// TwinCAT 3 PLC project PLC
// Title: Test PLC project for ads-client library
// Company: Jussi Isotalo
// Author: Jussi Isotalo
// Description: Copyright (c) 2022 Jussi Isotalo <j.isotalo91@gmail.com> Permission is hereby granted, free of charge, to any person obtaining a copy of this software and associated documentation files (the "Software"), to deal in the Software without restriction, including without limitation the rights to use, copy, modify, merge, publish, distribute, sublicense, and/or sell copies of the Software, and to permit persons to whom the Software is furnished to do so, subject to the following conditions: The above copyright notice and this permission notice shall be included in all copies or substantial portions of the Software. THE SOFTWARE IS PROVIDED "AS IS", WITHOUT WARRANTY OF ANY KIND, EXPRESS OR IMPLIED, INCLUDING BUT NOT LIMITED TO THE WARRANTIES OF MERCHANTABILITY, FITNESS FOR A PARTICULAR PURPOSE AND NONINFRINGEMENT. IN NO EVENT SHALL THE AUTHORS OR COPYRIGHT HOLDERS BE LIABLE FOR ANY CLAIM, DAMAGES OR OTHER LIABILITY, WHETHER IN AN ACTION OF CONTRACT, TORT OR OTHERWISE, ARISING FROM, OUT OF OR IN CONNECTION WITH THE SOFTWARE OR THE USE OR OTHER DEALINGS IN THE SOFTWARE
// ProgramVersion: 3.1.4023.0
// libraries:
//   Tc2_DataExchange, * (Beckhoff Automation GmbH)
//   Tc2_Standard, * (Beckhoff Automation GmbH)
//   Tc2_System, * (Beckhoff Automation GmbH)
//   Tc2_Utilities, * (Beckhoff Automation GmbH)
//   Tc3_Module, * (Beckhoff Automation GmbH)
// project tree:
//   AdsClientTests/Data types/ E_ExtendedEnum.TcDUT, FB_Block.TcPOU, FB_EmptyBlock.TcPOU, FB_EmptyBlock_1.TcPOU, I_Interface.TcIO, ST_Bits.TcDUT, ST_ComplexTypes_PackMode1.TcDUT, ST_ComplexTypes_PackMode8.TcDUT, ST_EmptyStruct.TcDUT, ST_IssueSpecificTypes.TcDUT, ST_SpecialTypes.TcDUT, ST_StandardTypes_PackMode1.TcDUT, ST_StandardTypes_PackMode8.TcDUT, ST_ComplexArrayTypes.TcDUT, ST_Struct.TcDUT, E_Enum.TcDUT, E_LintEnum.TcDUT, StandardTypesAlias.TcDUT, ST_StandardTypes.TcDUT, ST_StandardArrayTypes.TcDUT, ST_ComplexTypes.TcDUT, U_Union.TcDUT
//   AdsClientTests/ GVL_AdsClientTests.TcGVL, PRG_AdsClientTests.TcPOU
//   AdsClientTests/Read/ GVL_Read.TcGVL
//   AdsClientTests/RPC/ FB_Rpc.TcPOU, GVL_RPC.TcGVL
//   AdsClientTests/Subscription/ GVL_Subscription.TcGVL, PRG_Subscription.TcPOU
//   AdsClientTests/Symbols and datatypes/ GVL_SymbolsAndDataTypes.TcGVL, ST_TestDataType.TcDUT
//   AdsClientTests/Write/ GVL_Write.TcGVL
//   AdsClientTests/_OLD/ ST_Issue94.TcDUT, ST_Issue94_Byte.TcDUT, ST_PackMode1.TcDUT, ST_PackMode8.TcDUT, ST_Struct2.TcDUT
//   / PlcTask.TcTTO
// real-time tasks:
//   TASK PlcTask: cycle T#10ms, priority 20, ADS port 350
//   TASK PlcTask_852: cycle T#10ms, priority 21, ADS port 351

CONFIGURATION PLC
    RESOURCE PLC ON TwinCAT3
        TASK PlcTask(INTERVAL := T#10ms, PRIORITY := 20);
        PROGRAM PRG_AdsClientTests WITH PlcTask : PRG_AdsClientTests;
    END_RESOURCE
END_CONFIGURATION

// ---- AdsClientTests/Data types/E_ExtendedEnum.TcDUT
{attribute 'qualified_only'}
//{attribute 'strict'}
//This enum works differently than E_Enum only on TC 4026 and newer (comments and attributes)
TYPE E_ExtendedEnum :
(
	Disabled 	:= 0, //Machine is disabled
	Starting 	:= 50, //Machine is starting
	Running 	:= 100, //Machine is running
	Stopping	:= 200, //Machine is stopping
	
	{attribute 'ads-client-enum-attribute' := 'example-enum-value-ääö'}
	Unknown		:= -99 //Machine is ääöööÄÄÖö
);
END_TYPE

// ---- AdsClientTests/Data types/ST_Bits.TcDUT
TYPE ST_Bits :
STRUCT
	Bit_0 : BIT := TRUE;
	Bit_1 : BIT := FALSE;
	Bit_2 : BIT := FALSE;
	Bit_3 : BIT := TRUE;
	Bit_4 : BIT := TRUE;
	Bit_5 : BIT := FALSE;
	Bit_6 : BIT := FALSE;
	Bit_7 : BIT := TRUE;
	
	Bit_8 : BIT := FALSE;
	Bit_9 : BIT := TRUE;
	Bit_10 : BIT := TRUE;
	Bit_11 : BIT := FALSE;
	Bit_12 : BIT := FALSE;
	Bit_13 : BIT := TRUE;
	Bit_14 : BIT := TRUE;
	Bit_15 : BIT := FALSE;
	
	REAL_ : REAL := 3.14;
	
	Bit_16 : BIT := TRUE;
	Bit_17 : BIT := TRUE;
	Bit_18 : BIT := FALSE;
	Bit_19 : BIT := TRUE;
	Bit_20 : BIT := TRUE;
	Bit_21 : BIT := FALSE;
	Bit_22 : BIT := FALSE;
	Bit_23 : BIT := TRUE;
	
	Bit_24 : BIT := TRUE;
	Bit_25 : BIT := FALSE;
	Bit_26 : BIT := TRUE;
	Bit_27 : BIT := TRUE;
	Bit_28 : BIT := FALSE;
	Bit_29 : BIT := TRUE;
	Bit_30 : BIT := TRUE;
	Bit_31 : BIT := FALSE;
	
	Bit_32 : BIT := TRUE;
END_STRUCT
END_TYPE

// ---- AdsClientTests/Data types/ST_ComplexTypes_PackMode1.TcDUT
{attribute 'pack_mode' := '1'}
TYPE ST_ComplexTypes_PackMode1 :
STRUCT
	STRUCT_ 	: ST_StandardTypes;
	STRUCT_2 	: ST_StandardArrayTypes;
	ALIAS_ 		: StandardTypesAlias;
	ENUM_		: E_Enum := E_Enum.Running;
	ENUM_2		: E_Enum := E_Enum.Unknown;
	ENUM_3		: E_Enum := 5555; //Not a valid value
	ENUM_4		: E_LintEnum := E_LintEnum.Negative;
	ENUM_5		: (Implicit, Enum, Values, Go, Here) := Values;
	POINTER_	: POINTER TO ST_StandardTypes;
	REFERENCE_	: REFERENCE TO ST_StandardTypes;
	SUBRANGE_	: INT(-4095..4095) := 1234;
	UNION_		: U_Union := (STRING_ := 'A test string ääöö!!@@'); 
	UNION_2		: U_Union := (INT_ := 32767); 
	UNION_3		: U_Union := (REAL_ := 3.14);
	BLOCK_		: FB_Block;
	BLOCK_2		: TON := (PT := T#2S500MS);
	BLOCK_3		: TC2_System.FB_CreateDir := (sPathName := 'C:\Test');
	BLOCK_4		: Tc2_DataExchange.FB_ReadAdsSymByName := (sVarName := 'GVL_Test.Variable');
	INTERFACE_	: I_Interface := BLOCK_;
END_STRUCT
END_TYPE

// ---- AdsClientTests/Data types/ST_ComplexTypes_PackMode8.TcDUT
{attribute 'pack_mode' := '1'}
TYPE ST_ComplexTypes_PackMode8 :
STRUCT
	STRUCT_ 	: ST_StandardTypes;
	STRUCT_2 	: ST_StandardArrayTypes;
	ALIAS_ 		: StandardTypesAlias;
	ENUM_		: E_Enum := E_Enum.Running;
	ENUM_2		: E_Enum := E_Enum.Unknown;
	ENUM_3		: E_Enum := 5555; //Not a valid value
	ENUM_4		: E_LintEnum := E_LintEnum.Negative;
	ENUM_5		: (Implicit, Enum, Values, Go, Here) := Values;
	POINTER_	: POINTER TO ST_StandardTypes;
	REFERENCE_	: REFERENCE TO ST_StandardTypes;
	SUBRANGE_	: INT(-4095..4095) := 1234;
	UNION_		: U_Union := (STRING_ := 'A test string ääöö!!@@'); 
	UNION_2		: U_Union := (INT_ := 32767); 
	UNION_3		: U_Union := (REAL_ := 3.14);
	BLOCK_		: FB_Block;
	BLOCK_2		: TON := (PT := T#2S500MS);
	BLOCK_3		: TC2_System.FB_CreateDir := (sPathName := 'C:\Test');
	BLOCK_4		: Tc2_DataExchange.FB_ReadAdsSymByName := (sVarName := 'GVL_Test.Variable');
	INTERFACE_	: I_Interface := BLOCK_;
END_STRUCT
END_TYPE

// ---- AdsClientTests/Data types/ST_EmptyStruct.TcDUT
TYPE ST_EmptyStruct :
STRUCT
END_STRUCT
END_TYPE

// ---- AdsClientTests/Data types/ST_IssueSpecificTypes.TcDUT
TYPE ST_IssueSpecificTypes :
STRUCT
	Issue94	: ST_Issue94;
END_STRUCT
END_TYPE

// ---- AdsClientTests/Data types/ST_SpecialTypes.TcDUT
TYPE ST_SpecialTypes :
STRUCT
	NegativeIndexArray		: ARRAY[-100..100] OF LREAL := [1.11, 99(0.0), 5.55, 99(0.0), 9.99];
	MultiDimensionalArray	: ARRAY[1..3, 1..2] OF BYTE := [1, 2, 3, 4, 5, 6];
	ArrayOfArrays			: ARRAY[1..3] OF ARRAY[1..2] OF SINT := [[-1, -2], [-3, -4], [-5, -6]];
	
	PackMode1		: ST_StandardTypes_PackMode1;
	PackMode1_2		: ST_ComplexTypes_PackMode1;
	PackMode8		: ST_StandardTypes_PackMode8;
	PackMode8_2		: ST_ComplexTypes_PackMode8;
	
	EmptyBlock		: FB_EmptyBlock;
	EmptyStruct		: ST_EmptyStruct;
	EmptyArray 		: ARRAY[0..-1] OF BOOL; //How is this even possible..?
	
	Bits			: ST_Bits;
	
    {attribute 'TcEncoding':='UTF-8'}
	STRING_UTF8		: STRING := 'A test string ääöö!!@@';
END_STRUCT
END_TYPE

// ---- AdsClientTests/Data types/ST_StandardTypes_PackMode1.TcDUT
{attribute 'pack_mode' := '1'}
TYPE ST_StandardTypes_PackMode1 :
STRUCT
	BOOL_ 	: BOOL := TRUE;
	BOOL_2 	: BOOL := FALSE;
	BYTE_ 	: BYTE := 255;
	WORD_ 	: WORD := 65535;
	DWORD_ 	: DWORD := 4294967295;
	SINT_ 	: SINT := 127;
	SINT_2 	: SINT := -128;
	USINT_ 	: USINT := 255;
	INT_ 	: INT := 32767;
	INT_2 	: INT := -32768;
	UINT_ 	: UINT := 65535;
	DINT_ 	: DINT := 2147483647;
	DINT_2 	: DINT := -2147483648;
	UDINT_ 	: UDINT := 4294967295;
	REAL_ 	: REAL := 3.4E38;
	REAL_2 	: REAL := -3.4E38;
	REAL_3 	: REAL := 75483.545;
	REAL_4 	: REAL := -75483.545;
	STRING_	: STRING := 'A test string ääöö!!@@';
	STRING_2: STRING(255) := 'Lorem ipsum dolor sit amet, consectetur adipiscing elit. Pellentesque bibendum mauris vel metus rutrum, sed gravida justo dignissim. Aenean et nisi cursus, auctor mi vel, posuere enim. Suspendisse ultricies mauris in finibus tristique. Nullam turpis duis.';
	DATE_ 	: DATE := D#2106-02-06;
	DT_ 	: DT := DT#2106-02-06-06:28:15;
	DT_2 	: DATE_AND_TIME := DT#2106-02-06-06:28:15;
	TOD_ 	: TOD := TO_TOD(4294967295);
	TOD_2 	: TIME_OF_DAY := TO_TOD(4294967295);
	TIME_ 	: TIME := T#49D17H2M47S295MS;
	LWORD_	: LWORD := 18446744073709551615;
	LINT_	: LINT := 9223372036854775807;
	LINT_2	: LINT := -9223372036854775808;
	ULINT_	: ULINT := 18446744073709551615;
	LREAL_ 	: LREAL := 1.7E308;
	LREAL_2 : LREAL := -1.7E308;
	LREAL_3 : REAL := 75483.545;
	LREAL_4 : REAL := -75483.545;
	WSTRING_: WSTRING := "A test wstring ääöö!!@@ ẞẟΔش";
	WSTRING_2: WSTRING(255) := "Lorem ipsum dolor sit amet, consectetur adipiscing elit. Pellentesque bibendum mauris vel metus rutrum, sed gravida justo dignissim. Aenean et nisi cursus, auctor mi vel, posuere enim. Suspendisse ultricies mauris in finibus tristique. Nullam turpis duis.";
	//LDATE_	: LDATE := LD#2554-7-21;
	//LDT_	: LDT := LDT#2554-7-21-23:34:33.709551615;
	//LTOD_	: LTOD := LTOD#23:59:59.999999999;
	LTIME_ 	: LTIME := LTIME#213503D23H34M33S709MS551US615NS;
END_STRUCT
END_TYPE

// ---- AdsClientTests/Data types/ST_StandardTypes_PackMode8.TcDUT
{attribute 'pack_mode' := '8'}
TYPE ST_StandardTypes_PackMode8:
STRUCT
	BOOL_ 	: BOOL := TRUE;
	BOOL_2 	: BOOL := FALSE;
	BYTE_ 	: BYTE := 255;
	WORD_ 	: WORD := 65535;
	DWORD_ 	: DWORD := 4294967295;
	SINT_ 	: SINT := 127;
	SINT_2 	: SINT := -128;
	USINT_ 	: USINT := 255;
	INT_ 	: INT := 32767;
	INT_2 	: INT := -32768;
	UINT_ 	: UINT := 65535;
	DINT_ 	: DINT := 2147483647;
	DINT_2 	: DINT := -2147483648;
	UDINT_ 	: UDINT := 4294967295;
	REAL_ 	: REAL := 3.4E38;
	REAL_2 	: REAL := -3.4E38;
	REAL_3 	: REAL := 75483.545;
	REAL_4 	: REAL := -75483.545;
	STRING_	: STRING := 'A test string ääöö!!@@';
	STRING_2: STRING(255) := 'Lorem ipsum dolor sit amet, consectetur adipiscing elit. Pellentesque bibendum mauris vel metus rutrum, sed gravida justo dignissim. Aenean et nisi cursus, auctor mi vel, posuere enim. Suspendisse ultricies mauris in finibus tristique. Nullam turpis duis.';
	DATE_ 	: DATE := D#2106-02-06;
	DT_ 	: DT := DT#2106-02-06-06:28:15;
	DT_2 	: DATE_AND_TIME := DT#2106-02-06-06:28:15;
	TOD_ 	: TOD := TO_TOD(4294967295);
	TOD_2 	: TIME_OF_DAY := TO_TOD(4294967295);
	TIME_ 	: TIME := T#49D17H2M47S295MS;
	LWORD_	: LWORD := 18446744073709551615;
	LINT_	: LINT := 9223372036854775807;
	LINT_2	: LINT := -9223372036854775808;
	ULINT_	: ULINT := 18446744073709551615;
	LREAL_ 	: LREAL := 1.7E308;
	LREAL_2 : LREAL := -1.7E308;
	LREAL_3 : REAL := 75483.545;
	LREAL_4 : REAL := -75483.545;
	WSTRING_: WSTRING := "A test wstring ääöö!!@@ ẞẟΔش";
	WSTRING_2: WSTRING(255) := "Lorem ipsum dolor sit amet, consectetur adipiscing elit. Pellentesque bibendum mauris vel metus rutrum, sed gravida justo dignissim. Aenean et nisi cursus, auctor mi vel, posuere enim. Suspendisse ultricies mauris in finibus tristique. Nullam turpis duis.";
	//LDATE_	: LDATE := LD#2554-7-21;
	//LDT_	: LDT := LDT#2554-7-21-23:34:33.709551615;
	//LTOD_	: LTOD := LTOD#23:59:59.999999999;
	LTIME_ 	: LTIME := LTIME#213503D23H34M33S709MS551US615NS;
END_STRUCT
END_TYPE

// ---- AdsClientTests/Data types/ST_ComplexArrayTypes.TcDUT
TYPE ST_ComplexArrayTypes :
STRUCT
	STRUCT_ 	: ARRAY[0..2] OF ST_StandardTypes;
	STRUCT_2 	: ARRAY[0..2] OF ST_StandardArrayTypes;
	ALIAS_ 		: ARRAY[0..2] OF StandardTypesAlias;
	ENUM_		: ARRAY[0..2] OF E_Enum := [E_Enum.Running, E_Enum.Disabled, E_Enum.Stopping];
	ENUM_2		: ARRAY[0..2] OF E_Enum := [E_Enum.Unknown, E_Enum.Disabled, E_Enum.Starting];
	ENUM_3		: ARRAY[0..2] OF E_Enum := [5555, 0, E_Enum.Unknown];
	ENUM_4		: ARRAY[0..2] OF E_LintEnum := [E_LintEnum.Negative, E_LintEnum.Zero, E_LintEnum.Positive];
	ENUM_5		: ARRAY[0..2] OF (Implicit, Enum, Values, Go, Here) := [2, 0, 4];
	POINTER_	: ARRAY[0..2] OF POINTER TO ST_StandardTypes;
	//REFERENCE_	: ARRAY[0..2] OF REFERENCE TO ST_StandardTypes;
	SUBRANGE_	: ARRAY[0..2] OF INT(-4095..4095) := [1234, 0, -1234];
	UNION_		: ARRAY[0..2] OF U_Union := [
		(STRING_ := 'A test string ääöö!!@@'),
		(INT_ := 32767),
		(REAL_ := 3.14)
	]; 
	BLOCK_		: ARRAY[0..2] OF FB_Block := [
		(StrValue := 'First'),
		(),
		(StrValue := 'Third')
	];
	BLOCK_2		: ARRAY[0..2] OF TON := [(PT := T#2S500MS), (), (PT := T#123S)];
	BLOCK_3		: ARRAY[0..2] OF TC2_System.FB_CreateDir := [
		(sPathName := 'C:\Test'),
		(),
		(sPathName := 'C:\AnotherTest')
	];
	BLOCK_4		: ARRAY[0..2] OF Tc2_DataExchange.FB_ReadAdsSymByName := [
		(sVarName := 'GVL_Test.Variable'),
		(),
		(sVarName := 'GVL_Test.AnotherVariable')
	];
	INTERFACE_	: ARRAY[0..2] OF I_Interface := [BLOCK_[0], 0, BLOCK_[2]];
END_STRUCT
END_TYPE

// ---- AdsClientTests/Data types/ST_Struct.TcDUT
TYPE ST_Struct :
STRUCT
	SomeText : STRING(50) := 'Hello ads-client';
	SomeReal : REAL := 3.14159265359;
	SomeDate : DT := DT#2020-4-13-12:25:33;
END_STRUCT
END_TYPE

// ---- AdsClientTests/Symbols and datatypes/ST_TestDataType.TcDUT
{attribute 'pack_mode' := '3'}
{attribute 'ads-client-datatype-attribute' := 'example-datatype-value-ääö'}
//Test comment äääöö 
TYPE ST_TestDataType :
STRUCT
	Member : ST_Struct;
END_STRUCT
END_TYPE

// ---- AdsClientTests/Data types/E_Enum.TcDUT
{attribute 'qualified_only'}
//{attribute 'strict'}
TYPE E_Enum :
(
	Disabled 	:= 0,
	Starting 	:= 50,
	Running 	:= 100,
	Stopping	:= 200,
	Unknown		:= -99
);
END_TYPE

// ---- AdsClientTests/Data types/E_LintEnum.TcDUT
{attribute 'qualified_only'}
//{attribute 'strict'}
TYPE E_LintEnum :
(
	Negative := -9223372036854775808,
	Zero := 0,
	Positive := 9223372036854775807
) LINT;
END_TYPE

// ---- AdsClientTests/Data types/StandardTypesAlias.TcDUT
TYPE StandardTypesAlias : ST_StandardTypes; END_TYPE

// ---- AdsClientTests/Data types/ST_StandardTypes.TcDUT
TYPE ST_StandardTypes :
STRUCT
	BOOL_ 	: BOOL := TRUE;
	BOOL_2 	: BOOL := FALSE;
	BYTE_ 	: BYTE := 255;
	WORD_ 	: WORD := 65535;
	DWORD_ 	: DWORD := 4294967295;
	SINT_ 	: SINT := 127;
	SINT_2 	: SINT := -128;
	USINT_ 	: USINT := 255;
	INT_ 	: INT := 32767;
	INT_2 	: INT := -32768;
	UINT_ 	: UINT := 65535;
	DINT_ 	: DINT := 2147483647;
	DINT_2 	: DINT := -2147483648;
	UDINT_ 	: UDINT := 4294967295;
	REAL_ 	: REAL := 3.4E38;
	REAL_2 	: REAL := -3.4E38;
	REAL_3 	: REAL := 75483.545;
	REAL_4 	: REAL := -75483.545;
	STRING_	: STRING := 'A test string ääöö!!@@';
	STRING_2: STRING(255) := 'Lorem ipsum dolor sit amet, consectetur adipiscing elit. Pellentesque bibendum mauris vel metus rutrum, sed gravida justo dignissim. Aenean et nisi cursus, auctor mi vel, posuere enim. Suspendisse ultricies mauris in finibus tristique. Nullam turpis duis.';
	DATE_ 	: DATE := D#2106-02-06;
	DT_ 	: DT := DT#2106-02-06-06:28:15;
	DT_2 	: DATE_AND_TIME := DT#2106-02-06-06:28:15;
	TOD_ 	: TOD := TO_TOD(4294967295);
	TOD_2 	: TIME_OF_DAY := TO_TOD(4294967295);
	TIME_ 	: TIME := T#49D17H2M47S295MS;
	LWORD_	: LWORD := 18446744073709551615;
	LINT_	: LINT := 9223372036854775807;
	LINT_2	: LINT := -9223372036854775808;
	ULINT_	: ULINT := 18446744073709551615;
	LREAL_ 	: LREAL := 1.7E308;
	LREAL_2 : LREAL := -1.7E308;
	LREAL_3 : REAL := 75483.545;
	LREAL_4 : REAL := -75483.545;
	WSTRING_: WSTRING := "A test wstring ääöö!!@@ ẞẟΔش";
	WSTRING_2: WSTRING(255) := "Lorem ipsum dolor sit amet, consectetur adipiscing elit. Pellentesque bibendum mauris vel metus rutrum, sed gravida justo dignissim. Aenean et nisi cursus, auctor mi vel, posuere enim. Suspendisse ultricies mauris in finibus tristique. Nullam turpis duis.";
	//LDATE_	: LDATE := LD#2554-7-21;
	//LDT_	: LDT := LDT#2554-7-21-23:34:33.709551615;
	//LTOD_	: LTOD := LTOD#23:59:59.999999999;
	LTIME_ 	: LTIME := LTIME#213503D23H34M33S709MS551US615NS;
END_STRUCT
END_TYPE

// ---- AdsClientTests/Data types/ST_StandardArrayTypes.TcDUT
TYPE ST_StandardArrayTypes :
STRUCT
	BOOL_ 	: ARRAY[0..2] OF BOOL := [TRUE, FALSE, TRUE];
	BOOL_2 	: ARRAY[0..2] OF BOOL := [FALSE, TRUE, FALSE];
	BYTE_ 	: ARRAY[0..2] OF BYTE := [255, 254, 0];
	WORD_ 	: ARRAY[0..2] OF WORD := [65535, 65534, 0];
	DWORD_ 	: ARRAY[0..2] OF DWORD := [4294967295, 4294967294, 0];
	SINT_ 	: ARRAY[0..2] OF SINT := [127, 126, 0];
	SINT_2 	: ARRAY[0..2] OF SINT := [-128, -127, 0];
	USINT_ 	: ARRAY[0..2] OF USINT := [255, 254, 0];
	INT_ 	: ARRAY[0..2] OF INT := [32767, 0, -32768];
	INT_2 	: ARRAY[0..2] OF INT := [-32768, 0, 32767];
	UINT_ 	: ARRAY[0..2] OF UINT := [65535, 65534, 0];
	DINT_ 	: ARRAY[0..2] OF DINT := [2147483647, 0, -2147483648];
	DINT_2 	: ARRAY[0..2] OF DINT := [-2147483648, 0, 2147483647];
	UDINT_ 	: ARRAY[0..2] OF UDINT := [4294967295, 4294967294, 0];
	REAL_ 	: ARRAY[0..2] OF REAL := [3.4E38, 0, -3.4E38];
	REAL_2 	: ARRAY[0..2] OF REAL := [-3.4E38, 0, 3.4E38];
	REAL_3 	: ARRAY[0..2] OF REAL := [75483.545, 0, -75483.545];
	REAL_4 	: ARRAY[0..2] OF REAL := [-75483.545, 0, 75483.545];
	STRING_	: ARRAY[0..2] OF STRING := ['A test string ääöö!!@@', '', 'String value'];
	STRING_2: ARRAY[0..2] OF STRING(255) := [
		'Lorem ipsum dolor sit amet, consectetur adipiscing elit. Pellentesque bibendum mauris vel metus rutrum, sed gravida justo dignissim. Aenean et nisi cursus, auctor mi vel, posuere enim. Suspendisse ultricies mauris in finibus tristique. Nullam turpis duis.',
		'',
		'Proin tempor diam a felis fermentum, id molestie tortor pharetra. Phasellus condimentum rhoncus ultrices. Suspendisse ultricies nec neque quis sodales. In molestie vestibulum nulla eu gravida. Morbi orci ipsum, gravida elementum eros non, egestas egestas.'];
	DATE_ 	: ARRAY[0..2] OF DATE := [D#2106-02-06, D#2106-02-05, TO_DATE(0)];
	DT_ 	: ARRAY[0..2] OF DT := [DT#2106-02-06-06:28:15, DT#2106-02-06-06:28:14, TO_DT(0)];
	DT_2 	: ARRAY[0..2] OF DATE_AND_TIME := [DT#2106-02-06-06:28:15, DT#2106-02-06-06:28:14, TO_DT(0)];
	TOD_ 	: ARRAY[0..2] OF TOD := [TO_TOD(4294967295), TO_TOD(4294967294), TO_TOD(0)];
	TOD_2 	: ARRAY[0..2] OF TIME_OF_DAY := [TO_TOD(4294967295), TO_TOD(4294967294), TO_TOD(0)];
	TIME_ 	: ARRAY[0..2] OF TIME := [T#49D17H2M47S295MS, T#49D17H2M47S294MS, T#0S];
	LWORD_	: ARRAY[0..2] OF LWORD := [18446744073709551615, 18446744073709551614, 0];
	LINT_	: ARRAY[0..2] OF LINT := [9223372036854775807, 0, -9223372036854775808];
	LINT_2	: ARRAY[0..2] OF LINT := [-9223372036854775808, 0, 9223372036854775807];
	ULINT_	: ARRAY[0..2] OF ULINT := [18446744073709551615, 18446744073709551614, 0];
	LREAL_ 	: ARRAY[0..2] OF LREAL := [1.7E308, 0, -1.7E308];
	LREAL_2 : ARRAY[0..2] OF LREAL := [-1.7E308, 0, 1.7E308];
	LREAL_3	: ARRAY[0..2] OF REAL := [75483.545, 0, -75483.545];
	LREAL_4	: ARRAY[0..2] OF REAL := [-75483.545, 0, 75483.545];
	WSTRING_: ARRAY[0..2] OF WSTRING := ["A test wstring ääöö!!@@ ẞẟΔش", "", "ẞẟΔ"];
	WSTRING_2: ARRAY[0..2] OF WSTRING(255) := [
		"Lorem ipsum dolor sit amet, consectetur adipiscing elit. Pellentesque bibendum mauris vel metus rutrum, sed gravida justo dignissim. Aenean et nisi cursus, auctor mi vel, posuere enim. Suspendisse ultricies mauris in finibus tristique. Nullam turpis duis.",
		"",
		"Proin tempor diam a felis fermentum, id molestie tortor pharetra. Phasellus condimentum rhoncus ultrices. Suspendisse ultricies nec neque quis sodales. In molestie vestibulum nulla eu gravida. Morbi orci ipsum, gravida elementum eros non, egestas egestas."
	];
	//LDATE_	: ARRAY[0..2] OF LDATE := [LD#2554-7-21];
	//LDT_	: ARRAY[0..2] OF LDT := [LDT#2554-7-21-23:34:33.709551615];
	//LTOD_	: ARRAY[0..2] OF LTOD := [LTOD#23:59:59.999999999];
	LTIME_ 	: ARRAY[0..2] OF LTIME := [LTIME#213503D23H34M33S709MS551US615NS, LTIME#213503D23H34M33S709MS551US614NS, LTIME#0S];
END_STRUCT
END_TYPE

// ---- AdsClientTests/Data types/ST_ComplexTypes.TcDUT
TYPE ST_ComplexTypes :
STRUCT
	STRUCT_ 	: ST_StandardTypes;
	STRUCT_2 	: ST_StandardArrayTypes;
	ALIAS_ 		: StandardTypesAlias;
	ENUM_		: E_Enum := E_Enum.Running;
	ENUM_2		: E_Enum := E_Enum.Unknown;
	ENUM_3		: E_Enum := 5555; //Not a valid value
	ENUM_4		: E_LintEnum := E_LintEnum.Negative;
	ENUM_5		: (Implicit, Enum, Values, Go, Here) := Values;
	ENUM_6		: E_ExtendedEnum := E_Enum.Unknown;
	POINTER_	: POINTER TO ST_StandardTypes;
	REFERENCE_	: REFERENCE TO ST_StandardTypes;
	SUBRANGE_	: INT(-4095..4095) := 1234;
	UNION_		: U_Union := (STRING_ := 'A test string ääöö!!@@'); 
	UNION_2		: U_Union := (INT_ := 32767); 
	UNION_3		: U_Union := (REAL_ := 3.14);
	BLOCK_		: FB_Block;
	BLOCK_2		: TON := (PT := T#2S500MS);
	BLOCK_3		: TC2_System.FB_CreateDir := (sPathName := 'C:\Test');
	BLOCK_4		: Tc2_DataExchange.FB_ReadAdsSymByName := (sVarName := 'GVL_Test.Variable');
	INTERFACE_	: I_Interface := BLOCK_;
END_STRUCT
END_TYPE

// ---- AdsClientTests/Data types/U_Union.TcDUT
TYPE U_Union :
UNION
	INT_	: INT;
	BOOL_	: BOOL;
	UDINT_	: UDINT;
	STRING_	: STRING;
	REAL_	: REAL;
END_UNION
END_TYPE

// ---- AdsClientTests/_OLD/ST_Issue94.TcDUT
TYPE ST_Issue94 :
STRUCT
	BoolValue 	: bool := TRUE;
	ArrayValue 	:  ARRAY [0..1] OF ST_Issue94_Byte := [(ByteValue := 1), (ByteValue := 2)];
END_STRUCT
END_TYPE

// ---- AdsClientTests/_OLD/ST_Issue94_Byte.TcDUT
TYPE ST_Issue94_Byte :
STRUCT
	ByteValue : byte;
END_STRUCT
END_TYPE

// ---- AdsClientTests/_OLD/ST_PackMode1.TcDUT
{attribute 'pack_mode' := '1'}
TYPE ST_PackMode1 :
STRUCT
	BoolValue 	: BOOL := TRUE;
	StringValue : STRING(27) := 'A string value';
	LrealValue 	: LREAL := 12321.3123123;
	BoolArray 	: ARRAY[1..5] OF BOOL;
	BlockArray 	: ARRAY[1..5] OF r_trig;
	LargeBlock 	: Tc2_System.FB_FileOpen := (sPathName := 'test_path');
END_STRUCT
END_TYPE

// ---- AdsClientTests/_OLD/ST_PackMode8.TcDUT
{attribute 'pack_mode' := '8'}
TYPE ST_PackMode8 :
STRUCT
	BoolValue 	: BOOL := TRUE;
	StringValue : STRING(27) := 'A string value';
	LrealValue 	: LREAL := 12321.3123123;
	BoolArray 	: ARRAY[1..5] OF BOOL;
	BlockArray 	: ARRAY[1..5] OF r_trig;
	LargeBlock 	: Tc2_System.FB_FileOpen := (sPathName := 'test_path');
END_STRUCT
END_TYPE

// ---- AdsClientTests/_OLD/ST_Struct2.TcDUT
TYPE ST_Struct2 :
STRUCT
	BoolValue 	: BOOL := TRUE;
	StringValue : STRING(27) := 'A string value';
	LrealValue 	: LREAL := 12321.3123123;
	BoolArray 	: ARRAY[1..5] OF BOOL := [TRUE, FALSE, TRUE, FALSE, TRUE];
	SubStruct	: ST_Struct;
END_STRUCT
END_TYPE

// ---- AdsClientTests/GVL_AdsClientTests.TcGVL
{attribute 'qualified_only'}
VAR_GLOBAL
	VERSION			: STRING := '2.0.0';
	IsReset 		: BOOL := TRUE;
	IsTestProject 	: BOOL := TRUE;
	IsRunning 		: BOOL;
	TestPointer 	: POINTER TO BOOL; //For 32/64bit check
	IsTc2 			: BOOL := FALSE;
END_VAR

// ---- AdsClientTests/Read/GVL_Read.TcGVL
{attribute 'qualified_only'}
VAR_GLOBAL
	StandardTypes 		: ST_StandardTypes;
	StandardArrays 		: ST_StandardArrayTypes;
	ComplexTypes		: ST_ComplexTypes := (
		POINTER_ 	:= ADR(StandardTypes),
		REFERENCE_ 	:= StandardTypes 
	);
	ComplexArrayTypes	: ST_ComplexArrayTypes;
	SpecialTypes		: ST_SpecialTypes;
	IssueSpecificTypes	: ST_IssueSpecificTypes;
	
	test : pvoid := ADR(SpecialTypes.EmptyBlock);
	test2 : FB_EmptyBlock_1;
	
END_VAR

// ---- AdsClientTests/RPC/GVL_RPC.TcGVL
{attribute 'qualified_only'}
VAR_GLOBAL
	RpcBlock : FB_Rpc;
	
END_VAR

// ---- AdsClientTests/Subscription/GVL_Subscription.TcGVL
{attribute 'qualified_only'}
VAR_GLOBAL
	NumericValue_10ms : INT;
	NumericValue_100ms : INT;
	NumericValue_1000ms : INT;
	Numericvalue_Constant : INT := 12245;
END_VAR

// ---- AdsClientTests/Symbols and datatypes/GVL_SymbolsAndDataTypes.TcGVL
{attribute 'qualified_only'}
VAR_GLOBAL PERSISTENT
    {attribute 'ads-client-attribute' := 'example-value-ääö'}; 
	TestSymbol : STRING(82) := 'Some test value'; //Test comment äääöö
	TestDataType : ST_TestDataType;
END_VAR

// ---- AdsClientTests/Write/GVL_Write.TcGVL
{attribute 'qualified_only'}
VAR_GLOBAL
	StandardTypes 		: ST_StandardTypes;
	StandardArrays 		: ST_StandardArrayTypes;
	ComplexTypes		: ST_ComplexTypes := (
		POINTER_ 	:= ADR(StandardTypes),
		REFERENCE_ 	:= StandardTypes 
	);
	ComplexArrayTypes	: ST_ComplexArrayTypes;
	SpecialTypes		: ST_SpecialTypes;
	IssueSpecificTypes	: ST_IssueSpecificTypes;
	
END_VAR

// ---- AdsClientTests/Data types/I_Interface.TcIO
INTERFACE I_Interface

END_INTERFACE

// ---- AdsClientTests/PRG_AdsClientTests.TcPOU
PROGRAM PRG_AdsClientTests
VAR
	InitDone : BOOL;
	
END_VAR

IF NOT GVL_AdsClientTests.IsRunning THEN
	MEMSET(ADR(GVL_Write.StandardTypes), 0, SIZEOF(GVL_Write.StandardTypes));
	MEMSET(ADR(GVL_Write.StandardTypes), 0, SIZEOF(GVL_Write.StandardArrays));
	MEMSET(ADR(GVL_Write.ComplexTypes), 0, SIZEOF(GVL_Write.ComplexTypes));
	MEMSET(ADR(GVL_Write.ComplexArrayTypes), 0, SIZEOF(GVL_Write.ComplexArrayTypes));
	MEMSET(ADR(GVL_Write.SpecialTypes), 0, SIZEOF(GVL_Write.SpecialTypes));
	MEMSET(ADR(GVL_Write.IssueSpecificTypes), 0, SIZEOF(GVL_Write.IssueSpecificTypes));
	
	GVL_Write.ComplexTypes.POINTER_ := ADR(GVL_Write.StandardTypes);
	GVL_Write.ComplexTypes.REFERENCE_ ref= GVL_Write.StandardTypes;
	
	GVL_AdsClientTests.IsRunning := TRUE;
END_IF

PRG_Subscription();

END_PROGRAM

// ---- AdsClientTests/Subscription/PRG_Subscription.TcPOU
PROGRAM PRG_Subscription
VAR
	tonUpdate10ms : ton;
	tonUpdate100ms : ton;
	tonUpdate1000ms : ton;
END_VAR

//-------------------
// 10 ms
//-------------------
tonUpdate10ms(
	IN := TRUE,
	PT := T#10MS
);

IF tonUpdate10ms.Q THEN
	GVL_Subscription.NumericValue_10ms := GVL_Subscription.NumericValue_10ms + 1;

	tonUpdate10ms(IN := FALSE);
	tonUpdate10ms(IN := TRUE);
END_IF

//-------------------
// 100 ms
//-------------------
tonUpdate100ms(
	IN := TRUE,
	PT := T#100MS
);

IF tonUpdate100ms.Q THEN
	GVL_Subscription.NumericValue_100ms := GVL_Subscription.NumericValue_100ms + 1;

	tonUpdate100ms(IN := FALSE);
	tonUpdate100ms(IN := TRUE);
END_IF

//-------------------
// 1000 ms
//-------------------
tonUpdate1000ms(
	IN := TRUE,
	PT := T#1000MS
);

IF tonUpdate1000ms.Q THEN
	GVL_Subscription.NumericValue_1000ms := GVL_Subscription.NumericValue_1000ms + 1;

	tonUpdate1000ms(IN := FALSE);
	tonUpdate1000ms(IN := TRUE);
END_IF

END_PROGRAM

// ---- AdsClientTests/Data types/FB_EmptyBlock_1.TcPOU
FUNCTION_BLOCK FB_EmptyBlock_1
VAR_INPUT
END_VAR
VAR_OUTPUT
END_VAR
VAR
	value : BOOL;
END_VAR

END_FUNCTION_BLOCK

// ---- AdsClientTests/RPC/FB_Rpc.TcPOU
{attribute 'ads-client-attribute' := 'example-value-ääö'}; 
FUNCTION_BLOCK FB_Rpc
VAR_INPUT
END_VAR
VAR_OUTPUT
END_VAR
VAR
END_VAR

{attribute 'TcRpcEnable'}
METHOD Calculator : BOOL
VAR_INPUT
	Value1	: REAL;
	Value2	: REAL;
END_VAR
VAR_OUTPUT
	Sum			: REAL;
	Product 	: REAL;
	Division	: REAL;
END_VAR
//Return TRUE if all success
Calculator := TRUE;

Sum := Value1 + Value2;
Product := Value1 * Value2;

IF Value2 <> 0 THEN
	Division := Value1 / Value2;
ELSE
	Division := 0;
	Calculator := FALSE;
END_IF
END_METHOD

{attribute 'TcRpcEnable'}
{attribute 'ads-client-attribute' := 'example-value-ääö'}; 
METHOD NoParameters
VAR_INPUT
END_VAR
END_METHOD

{attribute 'TcRpcEnable'}
METHOD Structs : ST_Struct
VAR_INPUT
	{attribute 'ads-client-attribute' := 'example-value-ääö'}; 
	Input	: ST_Struct;
END_VAR
Structs.SomeText := CONCAT('Response: ', Input.SomeText);
Structs.SomeReal := Input.SomeReal * 10.0;
Structs.SomeDate := Input.SomeDate + T#24H;
END_METHOD

END_FUNCTION_BLOCK

// ---- AdsClientTests/Data types/FB_Block.TcPOU
FUNCTION_BLOCK FB_Block IMPLEMENTS I_Interface
VAR_INPUT
END_VAR
VAR_OUTPUT
END_VAR
VAR
	StrValue : string;
	Data : ST_StandardTypes;
END_VAR

END_FUNCTION_BLOCK

// ---- AdsClientTests/Data types/FB_EmptyBlock.TcPOU
FUNCTION_BLOCK FB_EmptyBlock
VAR_INPUT
END_VAR
VAR_OUTPUT
END_VAR
VAR
END_VAR

END_FUNCTION_BLOCK
